Staubli VAL3: TYPEBOOL.pgx

public program typeBool(num pX, num pY, bool v_bView, string pStr)
  local string lStr
begin
  //---------------------------------
  //  S H O W   O N E   S T R I N G
  //---------------------------------
  // Display one message in the
  // user page if nView is true else
  // it display one empty string
  //
  // See type()
  //---------------------------------
  // Staubli copyright 2003
  //                By CDIA 13 11 18
  //[Public]-------------------------
  //
  if (v_bView==true)
    lStr=pStr
  else
    call strFillChr(pStr,lStr," ")
  endIf
  call type(pX,pY,lStr)
end
